// TIA Portal V19 export
TYPE "PPrf_A0301_0302_Assemblaggio"
// stored: Access Published
   STRUCT
      Trasporto : "PPrf_A0301_Trasporto";
      Ribaltatore : "PPrf_A0301_Ribaltatore";
      Bordatrice : "PPrf_A0302_Bordatrice";
      HU_Cytropack : Struct
         Target_PressureParegg : Real;   // Set pressione HU Cytropack per pareggiamento longitudinale
         Target_MaxSpeedLimit : Real;   // Set limite massimo velocità HU Cytropack per pareggiamento longitudinale
      END_STRUCT;
   END_STRUCT;
END_TYPE
